FUNCTION_BLOCK FB_HMI_PRESSURES EXTENDS FB_HMI_COMPONENT
VAR_INPUT
END_VAR
VAR_OUTPUT
END_VAR
VAR
END_VAR

END_FUNCTION_BLOCK

(* stored: Version 1.1.0.1, ProductVersion 3.1.4024.14
   POU FB_HMI_PRESSURES: Id {f4fcd2cf-5351-4206-a9d2-944f16ec2a39}, SpecialFunc None *)
